FUNCTION_BLOCK Test_TStreamAdd_Read_BYTE EXTENDS T_UnitTestBase
VAR
    Stream : T_Stream(StreamLength := 2);
END_VAR



Stream.Init(2);

Stream.Add_BYTE(123);
    
Assertion.AssertEquals_UDINT(
    Expected := 3,
    Actual := Stream.Position,
    VariableName := 'Stream.Position');
    
Stream.Seek(0);

Assertion.AssertEquals_BYTE(
    Expected := 123,
    Actual := Stream.Read_BYTE(),
    VariableName := 'Stream.Read_BYTE()');
    
Assertion.AssertEquals_UDINT(
    Expected := 3,
    Actual := Stream.Position,
    VariableName := 'Stream.Position');
    
    
TestFinished();

END_FUNCTION_BLOCK

(* stored: Version 1.1.0.1, ProductVersion 3.1.4024.6
   POU Test_TStreamAdd_Read_BYTE: Id {e2f83219-ac36-4c11-a18b-54f10c7081f6}, SpecialFunc None *)
